// TIA Portal V17 export
// export: Created 2025-03-05T08:02:46.228224Z, ExportSetting WithDefaults, DisplayName Totally Integrated Automation Portal, DisplayVersion V17 Update 8, DisplayName TIA Portal Openness, DisplayVersion V17 Update 8, DisplayName TIA Portal Version Control Interface, DisplayVersion V17, DisplayName SINAMICS Startdrive Advanced, DisplayVersion V17 SP2, DisplayName SINAMICS Startdrive G110M, G120, G120C, G120D, G120P, G115D, DisplayVersion V17 SP2, DisplayName SINAMICS Startdrive G130, G150, S120, S150, SINAMICS MV, S210, DisplayVersion V17 SP2, DisplayName STEP 7 Professional, DisplayVersion V17 Update 8, DisplayName SINUMERIK ONE STEP 7 Toolbox, DisplayVersion V17 Update 12, DisplayName SINUMERIK 840D sl STEP 7 Toolbox, DisplayVersion V17 Update 12, DisplayName STEP 7 Safety, DisplayVersion V17 Update 6, DisplayName WinCC Advanced, DisplayVersion V17 Update 8
FUNCTION "FC2100_GENERAL" : Void   // FC2100, LAD
{ S7_Optimized_Access := 'FALSE' }
AUTHOR : ETXETAR
VERSION : 1.0
// stored: AutoNumber false, IsIECCheckEnabled false, SetENOAutomatically false, UDAEnableTagReadback false
   VAR CONSTANT
      FC_NUMBER : DInt := 2100;   // FC NUMBER
   END_VAR
BEGIN

REGION Network 1: ALWAYS OFF
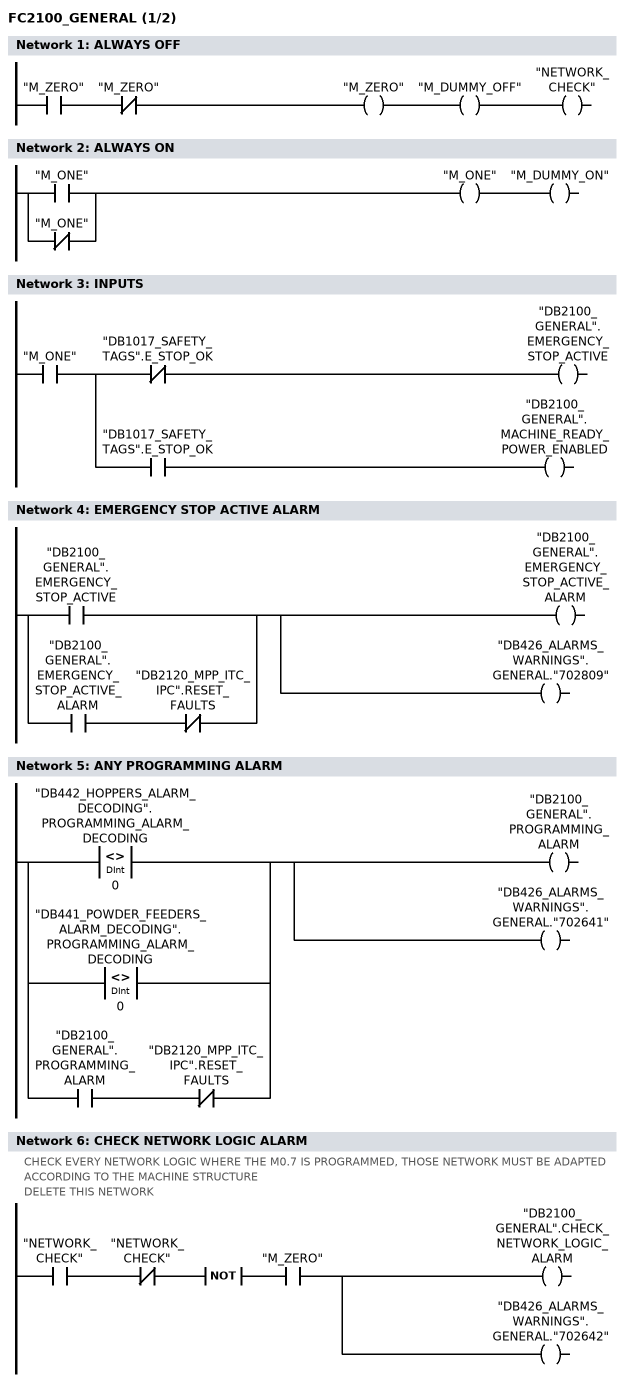
   RUNG wire#powerrail
      Contact( "M_ZERO" )
      I_Contact( "M_ZERO" )
      Coil( "M_ZERO" )
      Coil( "M_DUMMY_OFF" )
      Coil( "NETWORK_CHECK" )
   END_RUNG
   // the same network as SCL:
   "M_ZERO" := "M_ZERO" AND NOT "M_ZERO";
   "M_DUMMY_OFF" := "M_ZERO";
   "NETWORK_CHECK" := "M_ZERO";
END_REGION

REGION Network 2: ALWAYS ON
   RUNG wire#powerrail
      Contact( "M_ONE" )
      wire#w1
      Coil( "M_ONE" )
      Coil( "M_DUMMY_ON" )
   END_RUNG
   RUNG wire#powerrail
      I_Contact( "M_ONE" )
   END_RUNG wire#w1
   // the same network as SCL:
   "M_ONE" := "M_ONE" OR NOT "M_ONE";
   "M_DUMMY_ON" := "M_ONE";
END_REGION

REGION Network 3: INPUTS
   RUNG wire#powerrail
      Contact( "M_ONE" )
      wire#w1
      I_Contact( "DB1017_SAFETY_TAGS".E_STOP_OK )
      Coil( "DB2100_GENERAL".EMERGENCY_STOP_ACTIVE )
   END_RUNG
   RUNG wire#w1
      Contact( "DB1017_SAFETY_TAGS".E_STOP_OK )
      Coil( "DB2100_GENERAL".MACHINE_READY_POWER_ENABLED )
   END_RUNG
   // the same network as SCL:
   "DB2100_GENERAL".EMERGENCY_STOP_ACTIVE := "M_ONE" AND NOT "DB1017_SAFETY_TAGS".E_STOP_OK;
   "DB2100_GENERAL".MACHINE_READY_POWER_ENABLED := "M_ONE" AND "DB1017_SAFETY_TAGS".E_STOP_OK;
END_REGION

REGION Network 4: EMERGENCY STOP ACTIVE ALARM
   RUNG wire#powerrail
      Contact( "DB2100_GENERAL".EMERGENCY_STOP_ACTIVE )
      wire#w1
      Coil( "DB2100_GENERAL".EMERGENCY_STOP_ACTIVE_ALARM )
   END_RUNG
   RUNG wire#powerrail
      Contact( "DB2100_GENERAL".EMERGENCY_STOP_ACTIVE_ALARM )
      I_Contact( "DB2120_MPP_ITC_IPC".RESET_FAULTS )
   END_RUNG wire#w1
   RUNG wire#w1
      Coil( "DB426_ALARMS_WARNINGS".GENERAL."702809" )
   END_RUNG
   // the same network as SCL:
   "DB2100_GENERAL".EMERGENCY_STOP_ACTIVE_ALARM := "DB2100_GENERAL".EMERGENCY_STOP_ACTIVE OR ("DB2100_GENERAL".EMERGENCY_STOP_ACTIVE_ALARM AND NOT "DB2120_MPP_ITC_IPC".RESET_FAULTS);
   "DB426_ALARMS_WARNINGS".GENERAL."702809" := "DB2100_GENERAL".EMERGENCY_STOP_ACTIVE_ALARM;
END_REGION

REGION Network 5: ANY PROGRAMMING ALARM
   RUNG wire#powerrail
      { S7_Templates := "SrcType := DInt" } NE_Contact(in1 := "DB442_HOPPERS_ALARM_DECODING".PROGRAMMING_ALARM_DECODING, in2 := 0)
      wire#w1
      Coil( "DB2100_GENERAL".PROGRAMMING_ALARM )
   END_RUNG
   RUNG wire#powerrail
      { S7_Templates := "SrcType := DInt" } NE_Contact(in1 := "DB441_POWDER_FEEDERS_ALARM_DECODING".PROGRAMMING_ALARM_DECODING, in2 := 0)
   END_RUNG wire#w1
   RUNG wire#powerrail
      Contact( "DB2100_GENERAL".PROGRAMMING_ALARM )
      I_Contact( "DB2120_MPP_ITC_IPC".RESET_FAULTS )
   END_RUNG wire#w1
   RUNG wire#w1
      Coil( "DB426_ALARMS_WARNINGS".GENERAL."702641" )
   END_RUNG
   // the same network as SCL:
   "DB2100_GENERAL".PROGRAMMING_ALARM := ("DB442_HOPPERS_ALARM_DECODING".PROGRAMMING_ALARM_DECODING <> 0) OR ("DB441_POWDER_FEEDERS_ALARM_DECODING".PROGRAMMING_ALARM_DECODING <> 0) OR ("DB2100_GENERAL".PROGRAMMING_ALARM AND NOT "DB2120_MPP_ITC_IPC".RESET_FAULTS);
   "DB426_ALARMS_WARNINGS".GENERAL."702641" := "DB2100_GENERAL".PROGRAMMING_ALARM;
END_REGION

REGION Network 6: CHECK NETWORK LOGIC ALARM
   // CHECK EVERY NETWORK LOGIC WHERE THE M0.7 IS PROGRAMMED, THOSE NETWORK MUST BE ADAPTED ACCORDING TO THE MACHINE STRUCTURE
   // 
   // DELETE THIS NETWORK
   RUNG wire#powerrail
      Contact( "NETWORK_CHECK" )
      I_Contact( "NETWORK_CHECK" )
      Not()
      Contact( "M_ZERO" )
      wire#w1
      Coil( "DB2100_GENERAL".CHECK_NETWORK_LOGIC_ALARM )
   END_RUNG
   RUNG wire#w1
      Coil( "DB426_ALARMS_WARNINGS".GENERAL."702642" )
   END_RUNG
   // the same network as SCL:
   "DB2100_GENERAL".CHECK_NETWORK_LOGIC_ALARM := NOT ("NETWORK_CHECK" AND NOT "NETWORK_CHECK") AND "M_ZERO";
   "DB426_ALARMS_WARNINGS".GENERAL."702642" := "DB2100_GENERAL".CHECK_NETWORK_LOGIC_ALARM;
END_REGION

REGION Network 7: RESET PROGRAMMING ALARM
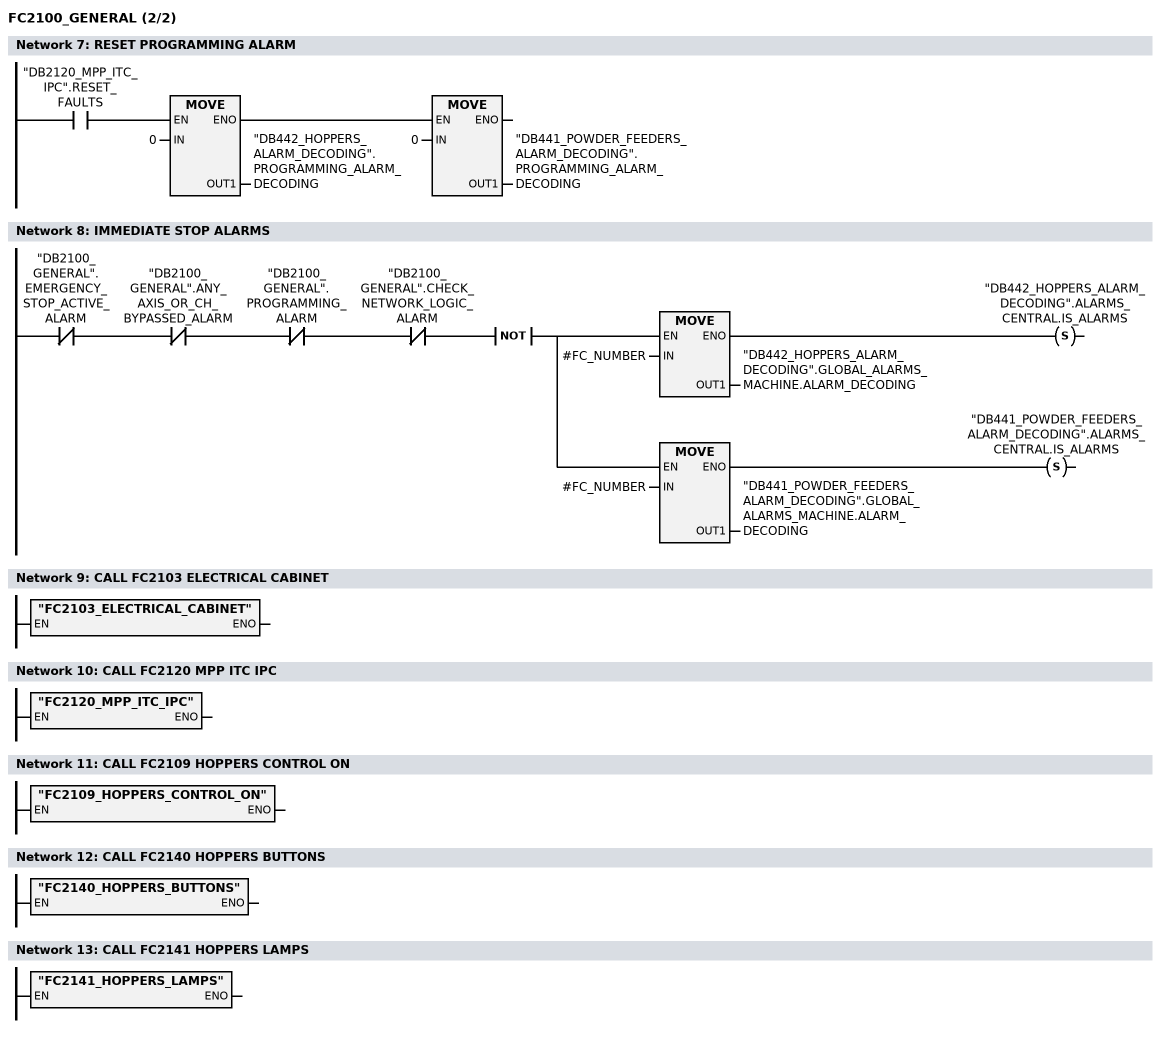
   RUNG wire#powerrail
      Contact( "DB2120_MPP_ITC_IPC".RESET_FAULTS )
      { S7_GenerateENO := "TRUE" } Move(in := 0, out1 => "DB442_HOPPERS_ALARM_DECODING".PROGRAMMING_ALARM_DECODING)
      { S7_GenerateENO := "TRUE" } Move(in := 0, out1 => "DB441_POWDER_FEEDERS_ALARM_DECODING".PROGRAMMING_ALARM_DECODING)
   END_RUNG
   // the same network as SCL:
   // ENO of a box is taken as its EN; it also drops when the box reports an error
   IF "DB2120_MPP_ITC_IPC".RESET_FAULTS THEN
       "DB442_HOPPERS_ALARM_DECODING".PROGRAMMING_ALARM_DECODING := 0;
       "DB441_POWDER_FEEDERS_ALARM_DECODING".PROGRAMMING_ALARM_DECODING := 0;
   END_IF;
END_REGION

REGION Network 8: IMMEDIATE STOP ALARMS
   RUNG wire#powerrail
      I_Contact( "DB2100_GENERAL".EMERGENCY_STOP_ACTIVE_ALARM )
      I_Contact( "DB2100_GENERAL".ANY_AXIS_OR_CH_BYPASSED_ALARM )
      I_Contact( "DB2100_GENERAL".PROGRAMMING_ALARM )
      I_Contact( "DB2100_GENERAL".CHECK_NETWORK_LOGIC_ALARM )
      Not()
      wire#w1
      { S7_GenerateENO := "TRUE" } Move(in := #FC_NUMBER, out1 => "DB442_HOPPERS_ALARM_DECODING".GLOBAL_ALARMS_MACHINE.ALARM_DECODING)
      S_Coil( "DB442_HOPPERS_ALARM_DECODING".ALARMS_CENTRAL.IS_ALARMS )
   END_RUNG
   RUNG wire#w1
      { S7_GenerateENO := "TRUE" } Move(in := #FC_NUMBER, out1 => "DB441_POWDER_FEEDERS_ALARM_DECODING".GLOBAL_ALARMS_MACHINE.ALARM_DECODING)
      S_Coil( "DB441_POWDER_FEEDERS_ALARM_DECODING".ALARMS_CENTRAL.IS_ALARMS )
   END_RUNG
   // the same network as SCL:
   // ENO of a box is taken as its EN; it also drops when the box reports an error
   IF NOT (NOT "DB2100_GENERAL".EMERGENCY_STOP_ACTIVE_ALARM AND NOT "DB2100_GENERAL".ANY_AXIS_OR_CH_BYPASSED_ALARM AND NOT "DB2100_GENERAL".PROGRAMMING_ALARM AND NOT "DB2100_GENERAL".CHECK_NETWORK_LOGIC_ALARM) THEN
       "DB442_HOPPERS_ALARM_DECODING".GLOBAL_ALARMS_MACHINE.ALARM_DECODING := #FC_NUMBER;
       "DB442_HOPPERS_ALARM_DECODING".ALARMS_CENTRAL.IS_ALARMS := TRUE;
       "DB441_POWDER_FEEDERS_ALARM_DECODING".GLOBAL_ALARMS_MACHINE.ALARM_DECODING := #FC_NUMBER;
       "DB441_POWDER_FEEDERS_ALARM_DECODING".ALARMS_CENTRAL.IS_ALARMS := TRUE;
   END_IF;
END_REGION

REGION Network 9: CALL FC2103 ELECTRICAL CABINET
   RUNG wire#powerrail
      "FC2103_ELECTRICAL_CABINET"()
   END_RUNG
   // the same network as SCL:
   "FC2103_ELECTRICAL_CABINET"();
END_REGION

REGION Network 10: CALL FC2120 MPP ITC IPC
   RUNG wire#powerrail
      "FC2120_MPP_ITC_IPC"()
   END_RUNG
   // the same network as SCL:
   "FC2120_MPP_ITC_IPC"();
END_REGION

REGION Network 11: CALL FC2109 HOPPERS CONTROL ON
   RUNG wire#powerrail
      "FC2109_HOPPERS_CONTROL_ON"()
   END_RUNG
   // the same network as SCL:
   "FC2109_HOPPERS_CONTROL_ON"();
END_REGION

REGION Network 12: CALL FC2140 HOPPERS BUTTONS
   RUNG wire#powerrail
      "FC2140_HOPPERS_BUTTONS"()
   END_RUNG
   // the same network as SCL:
   "FC2140_HOPPERS_BUTTONS"();
END_REGION

REGION Network 13: CALL FC2141 HOPPERS LAMPS
   RUNG wire#powerrail
      "FC2141_HOPPERS_LAMPS"()
   END_RUNG
   // the same network as SCL:
   "FC2141_HOPPERS_LAMPS"();
END_REGION
END_FUNCTION
